// TIA Portal V21 export
VAR_GLOBAL   // PLC tag table "KAllMotore"
END_VAR
VAR_GLOBAL CONSTANT   // user constants
   KAllMotore_Comunicazione : Int := 1;
   KAllMotore_DriveInAllarme : Int := 2;
   KAllMotore_Sovracorrente : Int := 3;
   KAllMotore_Coppia : Int := 4;
   KAllMotore_Termico : Int := 5;
   KAllMotore_TimeOutMarcia : Int := 6;
   KAllMotore_SezMotoreoreAperto : Int := 7;
   KAllMotore_ScattoTermicoServoventola : Int := 8;
   KAllMotore_RichiestaAzzeramento : Int := 9;
   KAllMotore_LimiteFisicoPosRaggiunto : Int := 10;
   KAllMotore_LimiteFisicoNegRaggiunto : Int := 11;
   KAllMotore_MotoreoreNonInAutoDaHmi : Int := 12;
   KAllMotore_MotoreoreNonInAutoDaPulsLoc : Int := 13;
   KAllMotore_FollowingError : Int := 14;
END_VAR
